(* Logix 5000 project; controller Lab5_FGBW vendor 1 type 14 code 92 rev 20.13; software revision 20.04 *)

TASK MainTask (continuous, watchdog 500 ms) : MainProgram

MODULES
   Local : vendor 1 type 14 code 92 (ICP 5, rev 20.13)
      DNET_Scanner : vendor 1 type 12 code 14 (ICP 11, rev 7.3, Output RPI 20 ms, Input RPI 20 ms)
END_MODULES

VAR_GLOBAL   (* controller tags *)
   Barcode_char : SINT[12];
   Barcode_Display : SINT[12];
   Barcode_Raw : STRING;
   DNET_MODE_Select_N : BOOL;
   Match_found_1 : SINT;
   New_Message_Sent_N : ALIAS FOR Local:11:I.Data[20].15;
   NO_LABEL : BOOL;
   NO_MATCH : BOOL;
   Prox_Sw : BOOL;
   Redi_Start_PB_N : ALIAS FOR Local:11:I.Data[15].1;
   RS_Start : BOOL;
   RS_Stop : BOOL;
   Run_mode : ALIAS FOR Local:11:O.CommandRegister.Run;
   Send_Next_Data_N : ALIAS FOR Local:11:O.Data[16].7;
   SIEO_1 : STRING;
   SIEO_2 : STRING;
   SIEO_3 : STRING;
   Tigger_Barcode_N : ALIAS FOR Local:11:O.Data[16].0;
   TIMER : TIMER[5] := ([0].PRE := 500, [1].PRE := 500);
   Trigger_PB : BOOL;
END_VAR

PROGRAM MainProgram   (* main routine MainRoutine *)
VAR
   DNET_MODE_Select : BOOL;   // Bit used to place Dnet in Run mode
   DNET_RUN_MODE : ALIAS FOR Local:11:O.CommandRegister.Run;   // DNET Scanner RUN Mode
   New_Message_Sent : ALIAS FOR Local:11:I.Data[75].15;   // Barcode New Message Being Sent Adaptascan Output 16
   Redi_Start_PB : ALIAS FOR Local:11:I.Data[72].1;   // Redi Station Start PB
   Send_Next_Data : ALIAS FOR Local:11:O.Data[75].7;   // Barcode Send Next Data Adaptascan Output 16
   Tigger_Barcode : ALIAS FOR Local:11:O.Data[75].0;   // Barcode Trigger to read label
END_VAR

ROUTINE DeviceNet   (* ladder *)
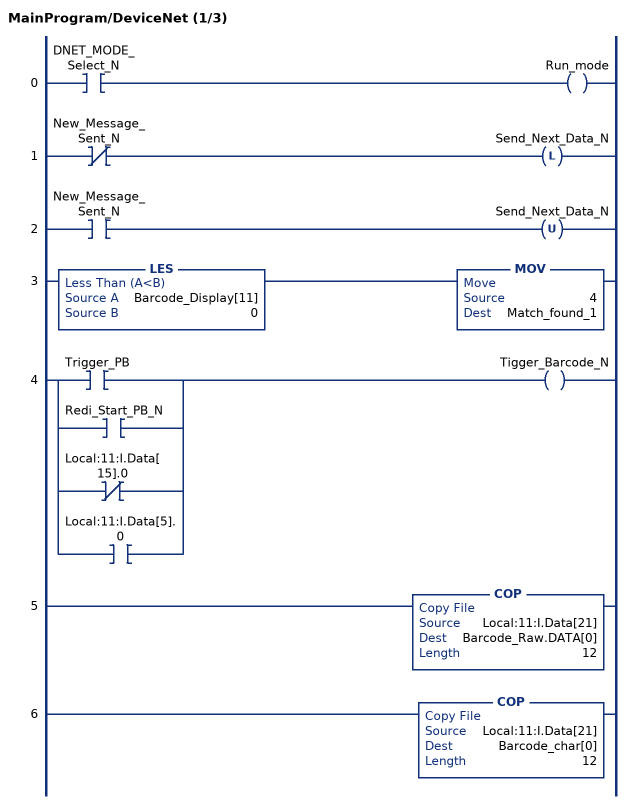
   0: XIC(DNET_MODE_Select_N)OTE(Run_mode);
   1: XIO(New_Message_Sent_N)OTL(Send_Next_Data_N);
   2: XIC(New_Message_Sent_N)OTU(Send_Next_Data_N);
   3: LES(Barcode_Display[11],0)MOV(4,Match_found_1);
   4: [XIC(Trigger_PB) ,XIC(Redi_Start_PB_N) ,XIO(Local:11:I.Data[15].0) ,XIC(Local:11:I.Data[5].0) ]OTE(Tigger_Barcode_N);
   5: COP(Local:11:I.Data[21],Barcode_Raw.DATA[0],12);
   6: COP(Local:11:I.Data[21],Barcode_char[0],12);
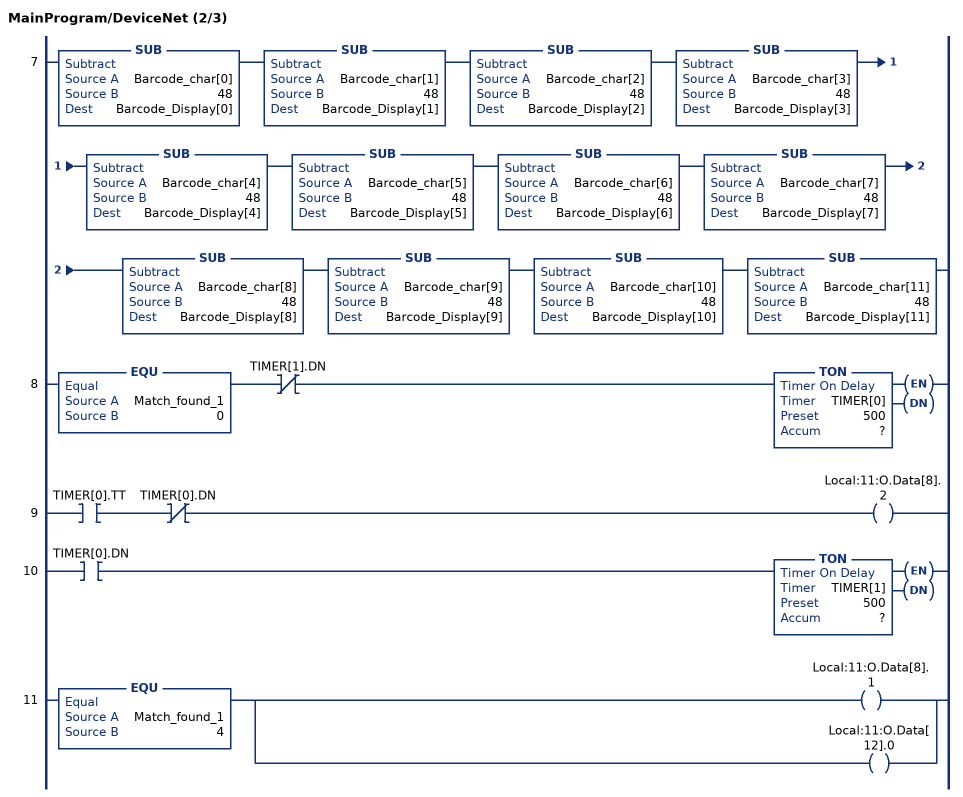
   7: SUB(Barcode_char[0],48,Barcode_Display[0])SUB(Barcode_char[1],48,Barcode_Display[1])SUB(Barcode_char[2],48,Barcode_Display[2])SUB(Barcode_char[3],48,Barcode_Display[3])SUB(Barcode_char[4],48,Barcode_Display[4])SUB(Barcode_char[5],48,Barcode_Display[5])SUB(Barcode_char[6],48,Barcode_Display[6])SUB(Barcode_char[7],48,Barcode_Display[7])SUB(Barcode_char[8],48,Barcode_Display[8])SUB(Barcode_char[9],48,Barcode_Display[9])SUB(Barcode_char[10],48,Barcode_Display[10])SUB(Barcode_char[11],48,Barcode_Display[11]);
   8: EQU(Match_found_1,0)XIO(TIMER[1].DN)TON(TIMER[0],?,?);
   9: XIC(TIMER[0].TT)XIO(TIMER[0].DN)OTE(Local:11:O.Data[8].2);
   10: XIC(TIMER[0].DN)TON(TIMER[1],?,?);
   11: EQU(Match_found_1,4)[OTE(Local:11:O.Data[8].1) ,OTE(Local:11:O.Data[12].0) ];
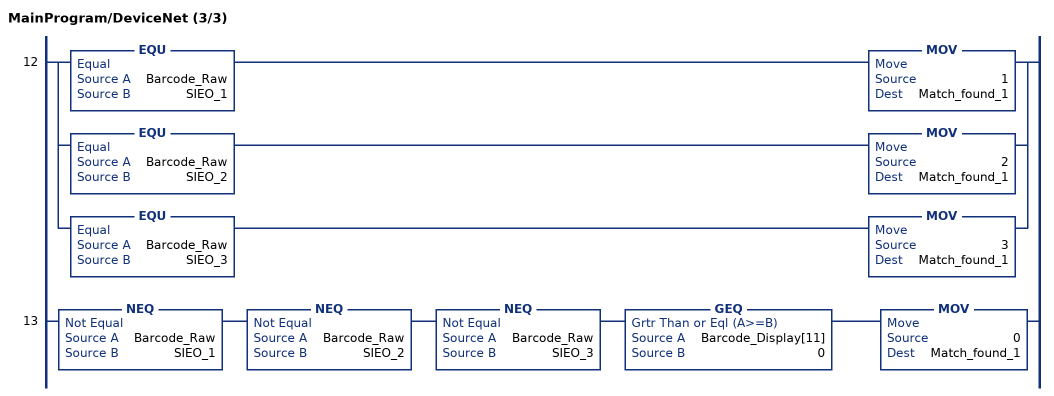
   12: [EQU(Barcode_Raw,SIEO_1) MOV(1,Match_found_1) ,EQU(Barcode_Raw,SIEO_2) MOV(2,Match_found_1) ,EQU(Barcode_Raw,SIEO_3) MOV(3,Match_found_1) ];
   13: NEQ(Barcode_Raw,SIEO_1)NEQ(Barcode_Raw,SIEO_2)NEQ(Barcode_Raw,SIEO_3)GEQ(Barcode_Display[11],0)MOV(0,Match_found_1);
END_ROUTINE

ROUTINE MainRoutine   (* ladder *)
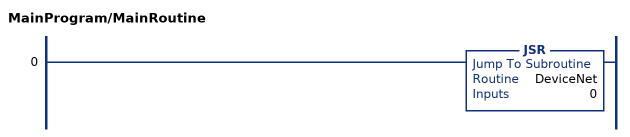
   0: JSR(DeviceNet,0);
END_ROUTINE
END_PROGRAM
